SUBAPPLICATION SystemTickSender_ISO (* SystemTick-Heartbeat auf einem VT-Zahlenfeld anzeigen (nur lokal, kein OPC-UA) *)
  (* Standard: 61499-2; Description: Copyright (c) 2026 Meisterschulen am Ostbahnhof This program and the accompanying materials are made available under the terms of the Eclipse Public License 2.0 which is available at https://www.eclipse.org/legal/epl-2.0/ SPDX-License-Identifier: EPL-2.0 *)
  (* Version 1.0, 2026-08-07, Franz Höpfinger, Meisterschulen am Ostbahnhof, initial API and implementation and/or initial documentation *)
  PACKAGE MyLib::sys;
  IMPORT isobus::UT::Q::const::IDs::ID_NULL;
  (* Documentation:
  SystemTick-Heartbeat auf einem VT-Zahlenfeld anzeigen
   Bündelt SystemTick mit der Anzeige auf dem lokalen VT: der laufende Tick-Zähler wird in ein VT-Zahlenausgabefeld (u16ObjId) geschrieben, damit man am Bildschirm auf einen Blick sieht, ob die Steuerung noch lebt (der Wert muss sich alle 200ms ändern).
   Funktionsbeschreibung
    - System_Tick liefert den Zählerstand als ADI (DINT).
   - ADI_TO_AUDI wandelt ihn in AUDI (UDINT) um, weil Q_NumericValue_AUDI (VT-Kommando "Change numeric value", Part 6 - F.22) einen vorzeichenlosen Wert erwartet.
    Rein lokal, ohne OPC-UA. Für zusätzliche Remote-Verteilung SystemTickSender_ISO_OPC, für ein Modul ohne eigene VT-Anbindung (nur OPC-UA) SystemTickSender_OPC verwenden.
  *)
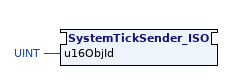
  VAR_INPUT
    u16ObjId : UINT := ID_NULL; (* Object ID VT-Zahlenausgabefeld (OutputNumberField), zeigt den Tick-Zaehlerstand an *)
  END_VAR
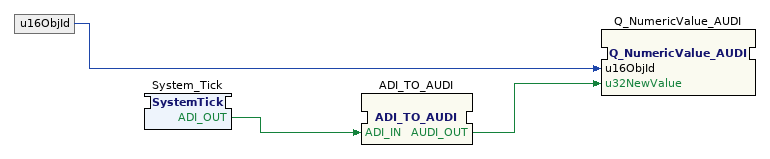
  FBS
    Q_NumericValue_AUDI : isobus::UT::Q::Q_NumericValue_AUDI;
    ADI_TO_AUDI : adapter::conversion::unidirectional::ADI_TO_AUDI;
  END_FBS
  SUBAPPS
    System_Tick : MyLib::sys::SystemTick;
  END_SUBAPPS
  DATA_CONNECTIONS
    u16ObjId TO Q_NumericValue_AUDI.u16ObjId;
  END_CONNECTIONS
  ADAPTER_CONNECTIONS
    ADI_TO_AUDI.AUDI_OUT TO Q_NumericValue_AUDI.u32NewValue;
    System_Tick.ADI_OUT TO ADI_TO_AUDI.ADI_IN;
  END_CONNECTIONS
END_SUBAPPLICATION
